FUNCTION_BLOCK delay (* Tamplate for a simple Basic Function Block Type *)
  (* Standard: 61499-2 *)
  (* Version 0.0, 2018-02-06, 4DIAC-IDE, 4DIAC-Consortium *)
  (* Version 1.0, 2016-05-26, AZ, fortiss GmbH *)
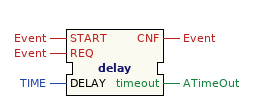
  EVENT_INPUT
    START;
    REQ; (* Normal Execution Request *)
  END_EVENT
  EVENT_OUTPUT
    CNF; (* Execution Confirmation *)
  END_EVENT
  VAR_INPUT
    DELAY : TIME;
  END_VAR
  PLUGS
    timeout : ATimeOut;
  END_PLUGS
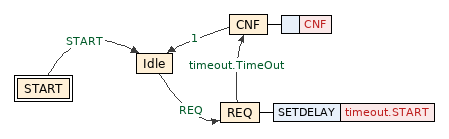
  EC_STATES
    START; (* Initial State *)
    Idle;
    REQ : SETDELAY -> timeout.START;
    CNF : -> CNF;
  END_STATES
  EC_TRANSITIONS
    START TO Idle := START;
    Idle TO REQ := REQ;
    REQ TO CNF := timeout.TimeOut;
    CNF TO Idle := 1;
  END_TRANSITIONS
  ALGORITHM SETDELAY IN ST: (* new algorithm *)
timeout.DT := DELAY;
  END_ALGORITHM
END_FUNCTION_BLOCK
